KUKA KRL program: wkz2_an.src, wkz2_an.dat

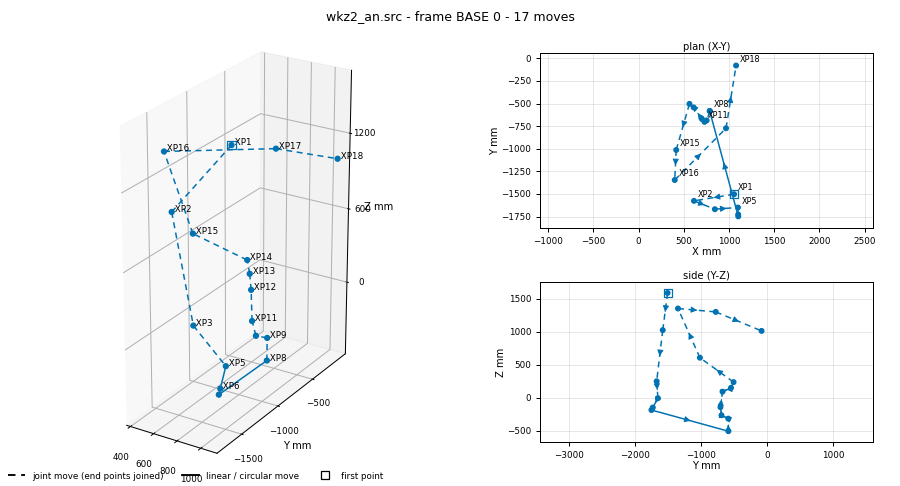
[picture p0: tool path of wkz2_an.src in frame BASE 0, 17 of 17 moves have a stored position in this frame; points joined in program order, loops and branches not executed]
--- wkz2_an.src ---
&ACCESS RVO2
&REL 264
&COMMENT PEGA_GRIPPER_ACTROS
&PARAM DISKPATH = Program/WKZ
DEF WKZ2_AN ( )

;FOLD INI
  ;FOLD BASISTECH INI
    GLOBAL INTERRUPT DECL 3 WHEN $STOPMESS==TRUE DO IR_STOPM ( )
    INTERRUPT ON 3
    BAS (#INITMOV,0 )
  ;ENDFOLD (BASISTECH INI)
  ;FOLD USER INI
    ;Make your modifications here
  ;ENDFOLD (USER INI)
;ENDFOLD (INI)
; Caracterização dos meios de produção:
; Versão Atual:10/06/2015
; Name: P13.090-R6 CHANGES: Pega Garra Actros

CHK_W8_Wechs_OK ( )          ; CHECK FLANGE OK
$ov_pro=50
;FOLD PTP P1 Vel=100 % PDAT1 Tool[8]:Tool Changer Base[0];%{PE}%R 8.2.24,%MKUKATPBASIS,%CMOVE,%VPTP,%P 1:PTP, 2:P1, 3:, 5:100, 7:PDAT1
$BWDSTART=FALSE
PDAT_ACT=PPDAT1
FDAT_ACT=FP1
BAS(#PTP_PARAMS,100)
PTP XP1
;ENDFOLD

;FOLD WAIT FOR ( IN 169 'DEPOSITO 2 OCUPADO' );%{PE}%R 8.2.24,%MKUKATPBASIS,%CEXT_WAIT_FOR,%VEXT_WAIT_FOR,%P 2:, 4:, 5:$IN, 6:169, 7:DEPOSITO 2 OCUPADO, 9:
WAIT FOR  ( $IN[169] )
;ENDFOLD
;FOLD WAIT FOR ( NOT IN 219 'PLACA DE SUPORTE FUNDIDA' );%{PE}%R 8.2.24,%MKUKATPBASIS,%CEXT_WAIT_FOR,%VEXT_WAIT_FOR,%P 2:, 4:NOT, 5:$IN, 6:219, 7:PLACA DE SUPORTE FUNDIDA, 9:
WAIT FOR  (  NOT $IN[219] )
;ENDFOLD
;FOLD PULSE 175 '' State=TRUE Time=0.3 sec;%{PE}%R 8.2.24,%MKUKATPBASIS,%COUT,%VPULSE,%P 2:175, 3:, 5:TRUE, 6:, 8:0.3
PULSE($OUT[175], TRUE,0.3)
;ENDFOLD

;FOLD PTP P2 Vel=100 % PDAT2 Tool[8]:Tool Changer Base[0];%{PE}%R 8.2.24,%MKUKATPBASIS,%CMOVE,%VPTP,%P 1:PTP, 2:P2, 3:, 5:100, 7:PDAT2
$BWDSTART=FALSE
PDAT_ACT=PPDAT2
FDAT_ACT=FP2
BAS(#PTP_PARAMS,100)
PTP XP2
;ENDFOLD

;FOLD WAIT FOR ( IN 173 'PROTECAO DE PINCA ABERTA' );%{PE}%R 8.2.24,%MKUKATPBASIS,%CEXT_WAIT_FOR,%VEXT_WAIT_FOR,%P 2:, 4:, 5:$IN, 6:173, 7:PROTECAO DE PINCA ABERTA, 9:
WAIT FOR  ( $IN[173] )
;ENDFOLD
;FOLD WAIT FOR ( NOT IN 174 'PROTECAO DE PINCA FECHADA' );%{PE}%R 8.2.24,%MKUKATPBASIS,%CEXT_WAIT_FOR,%VEXT_WAIT_FOR,%P 2:, 4:NOT, 5:$IN, 6:174, 7:PROTECAO DE PINCA FECHADA, 9:
WAIT FOR  (  NOT $IN[174] )
;ENDFOLD
;FOLD OUT 223 'DESBLOQUEIA MPS' State=FALSE ;%{PE}%R 8.2.24,%MKUKATPBASIS,%COUT,%VOUTX,%P 2:223, 3:DESBLOQUEIA MPS, 5:FALSE, 6:
$OUT[223]=FALSE
;ENDFOLD
;FOLD OUT 224 'BLOQUEIA MPS' State=TRUE ;%{PE}%R 8.2.24,%MKUKATPBASIS,%COUT,%VOUTX,%P 2:224, 3:BLOQUEIA MPS, 5:TRUE, 6:
$OUT[224]=TRUE
;ENDFOLD

;FOLD PTP P3 Vel=100 % PDAT3 Tool[8]:Tool Changer Base[0];%{PE}%R 8.2.24,%MKUKATPBASIS,%CMOVE,%VPTP,%P 1:PTP, 2:P3, 3:, 5:100, 7:PDAT3
$BWDSTART=FALSE
PDAT_ACT=PPDAT3
FDAT_ACT=FP3
BAS(#PTP_PARAMS,100)
PTP XP3
;ENDFOLD
;FOLD PTP P5 Vel=100 % PDAT5 Tool[8]:Tool Changer Base[0];%{PE}%R 8.2.24,%MKUKATPBASIS,%CMOVE,%VPTP,%P 1:PTP, 2:P5, 3:, 5:100, 7:PDAT5
$BWDSTART=FALSE
PDAT_ACT=PPDAT5
FDAT_ACT=FP5
BAS(#PTP_PARAMS,100)
PTP XP5
;ENDFOLD
;FOLD LIN P6 Vel=0.25 m/s CPDAT1 Tool[8]:Tool Changer Base[0];%{PE}%R 8.2.24,%MKUKATPBASIS,%CMOVE,%VLIN,%P 1:LIN, 2:P6, 3:, 5:0.25, 7:CPDAT1
$BWDSTART=FALSE
LDAT_ACT=LCPDAT1
FDAT_ACT=FP6
BAS(#CP_PARAMS,0.25)
LIN XP6
;ENDFOLD

;FOLD WAIT FOR ( IN 222 'KLASCHKA ATIVADO' );%{PE}%R 8.2.24,%MKUKATPBASIS,%CEXT_WAIT_FOR,%VEXT_WAIT_FOR,%P 2:, 4:, 5:$IN, 6:222, 7:KLASCHKA ATIVADO, 9:
WAIT FOR  ( $IN[222] )
;ENDFOLD
;FOLD OUT 223 'DESBLOQUEIA MPS' State=TRUE ;%{PE}%R 8.2.24,%MKUKATPBASIS,%COUT,%VOUTX,%P 2:223, 3:DESBLOQUEIA MPS, 5:TRUE, 6:
$OUT[223]=TRUE
;ENDFOLD
;FOLD OUT 224 'BLOQUEIA MPS' State=FALSE ;%{PE}%R 8.2.24,%MKUKATPBASIS,%COUT,%VOUTX,%P 2:224, 3:BLOQUEIA MPS, 5:FALSE, 6:
$OUT[224]=FALSE
;ENDFOLD

;FOLD WAIT FOR ( IN 217 'MPS DESTRAVADO' );%{PE}%R 8.2.24,%MKUKATPBASIS,%CEXT_WAIT_FOR,%VEXT_WAIT_FOR,%P 2:, 4:, 5:$IN, 6:217, 7:MPS DESTRAVADO, 9:
WAIT FOR  ( $IN[217] )
;ENDFOLD
;FOLD WAIT FOR ( NOT IN 221 'MPS TRAVADO' );%{PE}%R 8.2.24,%MKUKATPBASIS,%CEXT_WAIT_FOR,%VEXT_WAIT_FOR,%P 2:, 4:NOT, 5:$IN, 6:221, 7:MPS TRAVADO, 9:
WAIT FOR  (  NOT $IN[221] )
;ENDFOLD

;FOLD ; Ponto de pega da ferramenta;%{PE}%R 8.2.24,%MKUKATPBASIS,%CCOMMENT,%VNORMAL,%P 2:Ponto  de  pega  da  ferramenta
;ENDFOLD
;FOLD LIN P7 Vel=0.1 m/s CPDAT2 Tool[8]:Tool Changer Base[0];%{PE}%R 8.2.24,%MKUKATPBASIS,%CMOVE,%VLIN,%P 1:LIN, 2:P7, 3:, 5:0.1, 7:CPDAT2
$BWDSTART=FALSE
LDAT_ACT=LCPDAT2
FDAT_ACT=FP7
BAS(#CP_PARAMS,0.1)
LIN XP7
;ENDFOLD

;FOLD WAIT FOR ( IN 219 'PLACA DE SUPORTE FUNDIDA' );%{PE}%R 8.2.24,%MKUKATPBASIS,%CEXT_WAIT_FOR,%VEXT_WAIT_FOR,%P 2:, 4:, 5:$IN, 6:219, 7:PLACA DE SUPORTE FUNDIDA, 9:
WAIT FOR  ( $IN[219] )
;ENDFOLD
;FOLD OUT 223 'DESBLOQUEIA MPS' State=FALSE ;%{PE}%R 8.2.24,%MKUKATPBASIS,%COUT,%VOUTX,%P 2:223, 3:DESBLOQUEIA MPS, 5:FALSE, 6:
$OUT[223]=FALSE
;ENDFOLD
;FOLD OUT 224 'BLOQUEIA MPS' State=TRUE ;%{PE}%R 8.2.24,%MKUKATPBASIS,%COUT,%VOUTX,%P 2:224, 3:BLOQUEIA MPS, 5:TRUE, 6:
$OUT[224]=TRUE
;ENDFOLD
;FOLD WAIT FOR ( NOT IN 217 'MPS DESTRAVADO' );%{PE}%R 8.2.24,%MKUKATPBASIS,%CEXT_WAIT_FOR,%VEXT_WAIT_FOR,%P 2:, 4:NOT, 5:$IN, 6:217, 7:MPS DESTRAVADO, 9:
WAIT FOR  (  NOT $IN[217] )
;ENDFOLD
;FOLD WAIT FOR ( IN 221 'MPS TRAVADO' );%{PE}%R 8.2.24,%MKUKATPBASIS,%CEXT_WAIT_FOR,%VEXT_WAIT_FOR,%P 2:, 4:, 5:$IN, 6:221, 7:MPS TRAVADO, 9:
WAIT FOR  ( $IN[221] )
;ENDFOLD
;FOLD WAIT Time=1 sec;%{PE}%R 8.2.24,%MKUKATPBASIS,%CWAIT,%VWAIT,%P 3:1
WAIT SEC 1
;ENDFOLD

;FOLD IBUS ON SEGMENT_4;%{PE}%R 8.2.24,%MKUKATPBASIS,%CIBUS,%VMAP,%P 2:#ON, 3:4
$IBUS_ON=IBUS_SEGMENT[4]
$IBUS_OFF=0
;ENDFOLD

;FOLD LIN P8 Vel=0.25 m/s CPDAT3 Tool[2]:Gripper Parabrisa Actro Base[0];%{PE}%R 8.2.24,%MKUKATPBASIS,%CMOVE,%VLIN,%P 1:LIN, 2:P8, 3:, 5:0.25, 7:CPDAT3
$BWDSTART=FALSE
LDAT_ACT=LCPDAT3
FDAT_ACT=FP8
BAS(#CP_PARAMS,0.25)
LIN XP8
;ENDFOLD

;FOLD WAIT FOR ( NOT IN 169 'DEPOSITO 2 OCUPADO' );%{PE}%R 8.2.24,%MKUKATPBASIS,%CEXT_WAIT_FOR,%VEXT_WAIT_FOR,%P 2:, 4:NOT, 5:$IN, 6:169, 7:DEPOSITO 2 OCUPADO, 9:
WAIT FOR  (  NOT $IN[169] )
;ENDFOLD
;FOLD WAIT FOR ( IN 219 'PLACA DE SUPORTE FUNDIDA' );%{PE}%R 8.2.24,%MKUKATPBASIS,%CEXT_WAIT_FOR,%VEXT_WAIT_FOR,%P 2:, 4:, 5:$IN, 6:219, 7:PLACA DE SUPORTE FUNDIDA, 9:
WAIT FOR  ( $IN[219] )
;ENDFOLD

;FOLD ; SETAR GRUPO DE GRAMPOS 1 A 4 CLOSE;%{PE}%R 8.2.24,%MKUKATPBASIS,%CCOMMENT,%VNORMAL,%P 2:SETAR  GRUPO  DE  GRAMPOS  1  A  4 CLOSE
;ENDFOLD
;FOLD SET GRP 1 State=CLO GDAT1;%{PE}%R 8.2.4,%MKUKATPGRP,%CGRP,%VGRP,%P 2:1, 4:1, 5:#NO, 6:GDAT1, 8:0, 10:0
H50(GRP,1,1,GGDAT1)
;ENDFOLD
;FOLD SET GRP 2 State=CLO GDAT2;%{PE}%R 8.2.4,%MKUKATPGRP,%CGRP,%VGRP,%P 2:2, 4:1, 5:#NO, 6:GDAT2, 8:0, 10:0
H50(GRP,2,1,GGDAT2)
;ENDFOLD
;FOLD SET GRP 3 State=CLO GDAT3;%{PE}%R 8.2.4,%MKUKATPGRP,%CGRP,%VGRP,%P 2:3, 4:1, 5:#NO, 6:GDAT3, 8:0, 10:0
H50(GRP,3,1,GGDAT3)
;ENDFOLD
;FOLD SET GRP 4 State=CLO GDAT4;%{PE}%R 8.2.4,%MKUKATPGRP,%CGRP,%VGRP,%P 2:4, 4:1, 5:#NO, 6:GDAT4, 8:0, 10:0
H50(GRP,4,1,GGDAT4)
;ENDFOLD

;FOLD ; CHECAR SE GRAMPOS ESTAO FECHADOS;%{PE}%R 8.2.24,%MKUKATPBASIS,%CCOMMENT,%VNORMAL,%P 2:CHECAR  SE  GRAMPOS  ESTAO  FECHADOS
;ENDFOLD
chk_w2_grp1_clo ()
chk_w2_grp2_clo ()
chk_w2_grp3_clo ()
chk_w2_grp4_clo ()

;FOLD PTP P9 Vel=50 % PDAT6 Tool[2]:Gripper Parabrisa Actro Base[0];%{PE}%R 8.2.24,%MKUKATPBASIS,%CMOVE,%VPTP,%P 1:PTP, 2:P9, 3:, 5:50, 7:PDAT6
$BWDSTART=FALSE
PDAT_ACT=PPDAT6
FDAT_ACT=FP9
BAS(#PTP_PARAMS,50)
PTP XP9
;ENDFOLD
;FOLD PTP P10 Vel=50 % PDAT7 Tool[2]:Gripper Parabrisa Actro Base[0];%{PE}%R 8.2.24,%MKUKATPBASIS,%CMOVE,%VPTP,%P 1:PTP, 2:P10, 3:, 5:50, 7:PDAT7
$BWDSTART=FALSE
PDAT_ACT=PPDAT7
FDAT_ACT=FP10
BAS(#PTP_PARAMS,50)
PTP XP10
;ENDFOLD
;FOLD PTP P11 Vel=50 % PDAT8 Tool[2]:Gripper Parabrisa Actro Base[0];%{PE}%R 8.2.24,%MKUKATPBASIS,%CMOVE,%VPTP,%P 1:PTP, 2:P11, 3:, 5:50, 7:PDAT8
$BWDSTART=FALSE
PDAT_ACT=PPDAT8
FDAT_ACT=FP11
BAS(#PTP_PARAMS,50)
PTP XP11
;ENDFOLD
;FOLD PTP P12 Vel=50 % PDAT9 Tool[2]:Gripper Parabrisa Actro Base[0];%{PE}%R 8.2.24,%MKUKATPBASIS,%CMOVE,%VPTP,%P 1:PTP, 2:P12, 3:, 5:50, 7:PDAT9
$BWDSTART=FALSE
PDAT_ACT=PPDAT9
FDAT_ACT=FP12
BAS(#PTP_PARAMS,50)
PTP XP12
;ENDFOLD
;FOLD PTP P13 Vel=50 % PDAT10 Tool[2]:Gripper Parabrisa Actro Base[0];%{PE}%R 8.2.24,%MKUKATPBASIS,%CMOVE,%VPTP,%P 1:PTP, 2:P13, 3:, 5:50, 7:PDAT10
$BWDSTART=FALSE
PDAT_ACT=PPDAT10
FDAT_ACT=FP13
BAS(#PTP_PARAMS,50)
PTP XP13
;ENDFOLD
;FOLD PTP P14 Vel=50 % PDAT11 Tool[2]:Gripper Parabrisa Actro Base[0];%{PE}%R 8.2.24,%MKUKATPBASIS,%CMOVE,%VPTP,%P 1:PTP, 2:P14, 3:, 5:50, 7:PDAT11
$BWDSTART=FALSE
PDAT_ACT=PPDAT11
FDAT_ACT=FP14
BAS(#PTP_PARAMS,50)
PTP XP14
;ENDFOLD
;FOLD PTP P15 Vel=50 % PDAT12 Tool[2]:Gripper Parabrisa Actro Base[0];%{PE}%R 8.2.24,%MKUKATPBASIS,%CMOVE,%VPTP,%P 1:PTP, 2:P15, 3:, 5:50, 7:PDAT12
$BWDSTART=FALSE
PDAT_ACT=PPDAT12
FDAT_ACT=FP15
BAS(#PTP_PARAMS,50)
PTP XP15
;ENDFOLD
;FOLD PTP P16 CONT Vel=50 % PDAT13 Tool[2]:Gripper Parabrisa Actro Base[0];%{PE}%R 8.2.24,%MKUKATPBASIS,%CMOVE,%VPTP,%P 1:PTP, 2:P16, 3:C_PTP, 5:50, 7:PDAT13
$BWDSTART=FALSE
PDAT_ACT=PPDAT13
FDAT_ACT=FP16
BAS(#PTP_PARAMS,50)
PTP XP16 C_PTP
;ENDFOLD
;FOLD PTP P17 CONT Vel=50 % PDAT14 Tool[2]:Gripper Parabrisa Actro Base[0];%{PE}%R 8.2.24,%MKUKATPBASIS,%CMOVE,%VPTP,%P 1:PTP, 2:P17, 3:C_PTP, 5:50, 7:PDAT14
$BWDSTART=FALSE
PDAT_ACT=PPDAT14
FDAT_ACT=FP17
BAS(#PTP_PARAMS,50)
PTP XP17 C_PTP
;ENDFOLD
;FOLD PTP P18 Vel=50 % PDAT15 Tool[2]:Gripper Parabrisa Actro Base[0];%{PE}%R 8.2.24,%MKUKATPBASIS,%CMOVE,%VPTP,%P 1:PTP, 2:P18, 3:, 5:50, 7:PDAT15
$BWDSTART=FALSE
PDAT_ACT=PPDAT15
FDAT_ACT=FP18
BAS(#PTP_PARAMS,50)
PTP XP18
;ENDFOLD

;FOLD ; SETAR GRUPO DE GRAMPOS 1 A 4 OPEN;%{PE}%R 8.2.24,%MKUKATPBASIS,%CCOMMENT,%VNORMAL,%P 2:SETAR  GRUPO  DE  GRAMPOS  1  A  4 OPEN
;ENDFOLD
;FOLD SET GRP 1 State=OPN GDAT5;%{PE}%R 8.2.4,%MKUKATPGRP,%CGRP,%VGRP,%P 2:1, 4:2, 5:#NO, 6:GDAT5, 8:0, 10:0
H50(GRP,1,2,GGDAT5)
;ENDFOLD
;FOLD SET GRP 2 State=OPN GDAT6;%{PE}%R 8.2.4,%MKUKATPGRP,%CGRP,%VGRP,%P 2:2, 4:2, 5:#NO, 6:GDAT6, 8:0, 10:0
H50(GRP,2,2,GGDAT6)
;ENDFOLD
;FOLD SET GRP 3 State=OPN GDAT7;%{PE}%R 8.2.4,%MKUKATPGRP,%CGRP,%VGRP,%P 2:3, 4:2, 5:#NO, 6:GDAT7, 8:0, 10:0
H50(GRP,3,2,GGDAT7)
;ENDFOLD
;FOLD SET GRP 4 State=OPN GDAT9;%{PE}%R 8.2.4,%MKUKATPGRP,%CGRP,%VGRP,%P 2:4, 4:2, 5:#NO, 6:GDAT9, 8:0, 10:0
H50(GRP,4,2,GGDAT9)
;ENDFOLD
$ov_pro=100
chk_w2_grp1_opn ()
chk_w2_grp2_opn ()
chk_w2_grp3_opn ()
chk_w2_grp4_opn ()

;FOLD WAIT FOR ( IN 3339 'AGUARDA AGV NA POSICAO' );%{PE}%R 8.2.24,%MKUKATPBASIS,%CEXT_WAIT_FOR,%VEXT_WAIT_FOR,%P 2:, 4:, 5:$IN, 6:3339, 7:AGUARDA AGV NA POSICAO, 9:
WAIT FOR  ( $IN[3339] )
;ENDFOLD

END

--- wkz2_an.dat ---
&ACCESS RVO2
&REL 264
&COMMENT PEGA_GRIPPER_ACTROS
&PARAM DISKPATH = Program/WKZ
DEFDAT  wkz2_an
;FOLD EXTERNAL DECLARATIONS;%{PE}%MKUKATPBASIS,%CEXT,%VCOMMON,%P
;FOLD BASISTECH EXT;%{PE}%MKUKATPBASIS,%CEXT,%VEXT,%P
EXT  BAS (BAS_COMMAND  :IN,REAL  :IN )
DECL INT SUCCESS
;ENDFOLD (BASISTECH EXT)
;FOLD USER EXT;%{E}%MKUKATPUSER,%CEXT,%VEXT,%P
;Make your modifications here
;ENDFOLD (USER EXT)
;ENDFOLD (EXTERNAL DECLARATIONS)

;# ============ START PATH : wkz2_an =============
DECL FDAT Fnew_wkz2_an_p44={TOOL_NO 8,BASE_NO 0,IPO_FRAME #BASE,POINT2[] " "}
DECL PDAT PP_OLP1={VEL 100.0,ACC 50.0,APO_DIST 0.0}
DECL E6POS Xnew_wkz2_an_p44={X 612.940979,Y -1576.12097,Z 1025.58899,A -56.8068008,B -30.1534004,C 157.338699,S 2,T 2}
DECL FDAT Fnew_wkz2_an_p16={TOOL_NO 8,BASE_NO 0,IPO_FRAME #BASE,POINT2[] " "}
DECL PDAT PP_OLP2={VEL 100.0,ACC 100.0,APO_DIST 0.0}
DECL E6POS Xnew_wkz2_an_p16={X 843.835999,Y -1668.32202,Z 250.856995,A -56.8068008,B -30.1534004,C 157.338699,S 2,T 2}
DECL FDAT Fnew_wkz2_an_p17={TOOL_NO 8,BASE_NO 0,IPO_FRAME #BASE,POINT2[] " "}
DECL PDAT PP_OLP3={VEL 100.0,ACC 100.0,APO_DIST 0.0}
DECL E6POS Xnew_wkz2_an_p17={X 1098.79395,Y -1649.33801,Z -5.05700016,A -73.2769012,B -27.9207001,C 173.073105,S 2,T 2}
DECL FDAT Fnew_wkz2_an_p4={TOOL_NO 8,BASE_NO 0,IPO_FRAME #BASE,POINT2[] " "}
DECL E6POS Xnew_wkz2_an_p4={X 1101.74304,Y -1726.75305,Z -146.546005,A -73.2770996,B -27.9211998,C 173.073196,S 2,T 2}
DECL LDAT LL_OLP1={VEL 0.25,ACC 100.0,APO_DIST 0.0,APO_FAC 0.0,ORI_TYP #VAR,CIRC_TYP #BASE,JERK_FAC 50.0}
DECL FDAT Fnew_wkz2_an_p5={TOOL_NO 8,BASE_NO 0,IPO_FRAME #BASE,POINT2[] " "}
DECL E6POS Xnew_wkz2_an_p5={X 1102.474,Y -1745.90198,Z -181.546005,A -73.2769012,B -27.9209003,C 173.073105,S 2,T 2}
DECL LDAT LL_OLP2={VEL 0.100000001,ACC 100.0,APO_DIST 0.0,APO_FAC 0.0,ORI_TYP #VAR,CIRC_TYP #BASE,JERK_FAC 50.0}
DECL FDAT Fnew_wkz2_an_p11={TOOL_NO 2,BASE_NO 0,IPO_FRAME #BASE,POINT2[] " "}
DECL E6POS Xnew_wkz2_an_p11={X 786.29303,Y -582.55603,Z -504.964996,A 0.253399998,B -1.02199996,C -179.584305,S 2,T 2}
DECL LDAT LL_OLP3={VEL 0.25,ACC 100.0,APO_DIST 0.0,APO_FAC 0.0,ORI_TYP #VAR,CIRC_TYP #BASE,JERK_FAC 50.0}
DECL FDAT Fnew_wkz2_an_p12={TOOL_NO 2,BASE_NO 0,IPO_FRAME #BASE,POINT2[] " "}
DECL PDAT PP_OLP4={VEL 100.0,ACC 50.0,APO_DIST 0.0}
DECL E6POS Xnew_wkz2_an_p12={X 788.83197,Y -583.976013,Z -314.804993,A 0.253100008,B -1.0223,C -179.584702,S 2,T 2}
DECL FDAT Fnew_wkz2_an_p13={TOOL_NO 2,BASE_NO 0,IPO_FRAME #BASE,POINT2[] " "}
DECL PDAT PP_OLP5={VEL 100.0,ACC 50.0,APO_DIST 0.0}
DECL E6POS Xnew_wkz2_an_p13={X 753.492004,Y -686.713989,Z -263.341003,A 0.255299985,B -1.02450001,C -179.584595,S 2,T 2}
DECL FDAT Fnew_wkz2_an_p18={TOOL_NO 2,BASE_NO 0,IPO_FRAME #BASE,POINT2[] " "}
DECL PDAT PP_OLP6={VEL 100.0,ACC 100.0,APO_DIST 0.0}
DECL E6POS Xnew_wkz2_an_p18={X 728.877991,Y -702.304993,Z -141.432007,A 0.00469999993,B -0.533699989,C -179.897705,S 2,T 2}
DECL FDAT Fnew_wkz2_an_p33={TOOL_NO 2,BASE_NO 0,IPO_FRAME #BASE,POINT2[] " "}
DECL PDAT PP_OLP7={VEL 100.0,ACC 100.0,APO_DIST 0.0}
DECL E6POS Xnew_wkz2_an_p33={X 702.591003,Y -670.484009,Z -1.97099996,A -0.302599996,B -1.01380002,C -179.617706,S 2,T 2}
DECL FDAT Fnew_wkz2_an_p37={TOOL_NO 2,BASE_NO 0,IPO_FRAME #BASE,POINT2[] " "}
DECL PDAT PP_OLP8={VEL 100.0,ACC 100.0,APO_DIST 0.0}
DECL E6POS Xnew_wkz2_an_p37={X 600.364014,Y -522.731018,Z 51.5839996,A -0.309100002,B -1.0122,C -179.757004,S 2,T 2}
DECL FDAT Fnew_wkz2_an_p38={TOOL_NO 2,BASE_NO 0,IPO_FRAME #BASE,POINT2[] " "}
DECL PDAT PP_OLP9={VEL 100.0,ACC 100.0,APO_DIST 0.0}
DECL E6POS Xnew_wkz2_an_p38={X 562.674011,Y -503.727997,Z 237.981003,A -9.11750031,B -5.62230015,C 153.765503,S 2,T 2}
DECL FDAT Fnew_wkz2_an_p42={TOOL_NO 2,BASE_NO 0,IPO_FRAME #BASE,POINT2[] " "}
DECL PDAT PP_OLP10={VEL 100.0,ACC 100.0,APO_DIST 0.0}
DECL E6POS Xnew_wkz2_an_p42={X 978.356018,Y -287.113007,Z 541.031982,A 9.17619991,B -20.1103001,C 143.3797,S 2,T 2}
DECL FDAT Fnew_wkz2_an_p43={TOOL_NO 2,BASE_NO 0,IPO_FRAME #BASE,POINT2[] " "}
DECL PDAT PP_OLP11={VEL 100.0,ACC 100.0,APO_DIST 0.0}
DECL E6POS Xnew_wkz2_an_p43={X 1078.0,Y -78.862999,Z 664.578003,A 0.512600005,B -24.8574009,C 146.008606,S 2,T 2}
DECL BASIS_SUGG_T LAST_BASIS={POINT1[] "P20                     ",POINT2[] "P20                     ",CP_PARAMS[] "CPDAT3                  ",PTP_PARAMS[] "PDAT17                  ",CONT[] "                        ",CP_VEL[] "0.25                    ",PTP_VEL[] "100                     ",SYNC_PARAMS[] "SYNCDAT                 ",SPL_NAME[] "S0                      "}
DECL E6POS XP1={X 1055.88904,Y -1502.42297,Z 1588.46497,A -71.8623123,B -60.8086586,C 178.730499,S 18,T 2,E1 0.0,E2 0.0,E3 0.0,E4 0.0,E5 0.0,E6 0.0}
DECL FDAT FP1={TOOL_NO 8,BASE_NO 0,IPO_FRAME #BASE,POINT2[] " ",TQ_STATE FALSE}
DECL PDAT PPDAT1={VEL 100.0,ACC 100.0,APO_DIST 100.0,GEAR_JERK 50.0}
DECL E6POS XP2={X 612.938782,Y -1576.11304,Z 1025.57605,A -56.8084106,B -30.1530895,C 157.339798,S 18,T 2,E1 0.0,E2 0.0,E3 0.0,E4 0.0,E5 0.0,E6 0.0}
DECL FDAT FP2={TOOL_NO 8,BASE_NO 0,IPO_FRAME #BASE,POINT2[] " ",TQ_STATE FALSE}
DECL PDAT PPDAT2={VEL 100.0,ACC 100.0,APO_DIST 100.0,GEAR_JERK 50.0}
DECL E6POS XP3={X 843.833618,Y -1668.31494,Z 250.858704,A -56.807251,B -30.1531506,C 157.339203,S 18,T 2,E1 0.0,E2 0.0,E3 0.0,E4 0.0,E5 0.0,E6 0.0}
DECL FDAT FP3={TOOL_NO 8,BASE_NO 0,IPO_FRAME #BASE,POINT2[] " ",TQ_STATE FALSE}
DECL PDAT PPDAT3={VEL 100.0,ACC 50.0,APO_DIST 100.0,GEAR_JERK 50.0}
DECL E6POS XP4={X 1070.15295,Y -1848.78406,Z 103.901703,A -73.2903366,B -27.8212204,C 173.081299,S 18,T 2,E1 0.0,E2 0.0,E3 0.0,E4 0.0,E5 0.0,E6 0.0}
DECL FDAT FP4={TOOL_NO 8,BASE_NO 0,IPO_FRAME #BASE,POINT2[] " ",TQ_STATE FALSE}
DECL PDAT PPDAT4={VEL 100.0,ACC 100.0,APO_DIST 100.0,GEAR_JERK 50.0}
DECL GRP_SUGG_T LAST_GRP={NUMBER[] "4                       ",STATE[] "1                       ",PARAMS[] "GDAT4                   "}
DECL E6POS XP5={X 1098.79602,Y -1649.34802,Z -5.03718805,A -73.2673264,B -27.9203205,C 173.069504,S 18,T 2,E1 0.0,E2 0.0,E3 0.0,E4 0.0,E5 0.0,E6 0.0}
DECL FDAT FP5={TOOL_NO 8,BASE_NO 0,IPO_FRAME #BASE,POINT2[] " ",TQ_STATE FALSE}
DECL PDAT PPDAT5={VEL 100.0,ACC 100.0,APO_DIST 100.0,GEAR_JERK 50.0}
DECL E6POS XP6={X 1101.74097,Y -1726.75598,Z -146.535294,A -73.2780228,B -27.9206905,C 173.074005,S 18,T 2,E1 0.0,E2 0.0,E3 0.0,E4 0.0,E5 0.0,E6 0.0}
DECL FDAT FP6={TOOL_NO 8,BASE_NO 0,IPO_FRAME #BASE,POINT2[] " ",TQ_STATE FALSE}
DECL LDAT LCPDAT1={VEL 2.0,ACC 100.0,APO_DIST 100.0,APO_FAC 50.0,AXIS_VEL 100.0,AXIS_ACC 100.0,ORI_TYP #VAR,CIRC_TYP #BASE,JERK_FAC 50.0,GEAR_JERK 50.0,EXAX_IGN 0}
DECL E6POS XP7={X 1102.50403,Y -1747.31702,Z -184.174393,A -73.2694321,B -27.9181194,C 173.068497,S 18,T 2,E1 0.0,E2 0.0,E3 0.0,E4 0.0,E5 0.0,E6 0.0}
DECL FDAT FP7={TOOL_NO 8,BASE_NO 0,IPO_FRAME #BASE,POINT2[] " ",TQ_STATE FALSE}
DECL LDAT LCPDAT2={VEL 2.0,ACC 100.0,APO_DIST 100.0,APO_FAC 50.0,AXIS_VEL 100.0,AXIS_ACC 100.0,ORI_TYP #VAR,CIRC_TYP #BASE,JERK_FAC 50.0,GEAR_JERK 50.0,EXAX_IGN 0}
DECL E6POS XP8={X 786.28833,Y -582.550781,Z -504.954407,A 0.253419489,B -1.02197099,C -179.584,S 18,T 2,E1 0.0,E2 0.0,E3 0.0,E4 0.0,E5 0.0,E6 0.0}
DECL FDAT FP8={TOOL_NO 2,BASE_NO 0,IPO_FRAME #BASE,POINT2[] " ",TQ_STATE FALSE}
DECL LDAT LCPDAT3={VEL 2.0,ACC 100.0,APO_DIST 100.0,APO_FAC 50.0,AXIS_VEL 100.0,AXIS_ACC 100.0,ORI_TYP #VAR,CIRC_TYP #BASE,JERK_FAC 50.0,GEAR_JERK 50.0,EXAX_IGN 0}
DECL E6POS XP9={X 788.821777,Y -583.967224,Z -314.793488,A 0.253417194,B -1.02216303,C -179.584198,S 18,T 2,E1 0.0,E2 0.0,E3 0.0,E4 0.0,E5 0.0,E6 0.0}
DECL FDAT FP9={TOOL_NO 2,BASE_NO 0,IPO_FRAME #BASE,POINT2[] " ",TQ_STATE FALSE}
DECL PDAT PPDAT6={VEL 100.0,ACC 100.0,APO_DIST 100.0,GEAR_JERK 50.0}
DECL GRP_TYP GCONT={G_APO #YES,GRP_TIME 0.0,CTRL #OFF,DLY 0,DST 0}
DECL E6POS XP10={X 753.30658,Y -686.742981,Z -263.305695,A 0.262432188,B -1.01997399,C -179.584,S 18,T 2,E1 0.0,E2 0.0,E3 0.0,E4 0.0,E5 0.0,E6 0.0}
DECL FDAT FP10={TOOL_NO 2,BASE_NO 0,IPO_FRAME #BASE,POINT2[] " ",TQ_STATE FALSE}
DECL PDAT PPDAT7={VEL 100.0,ACC 50.0,APO_DIST 100.0,GEAR_JERK 50.0}
DECL E6POS XP11={X 728.857788,Y -702.299377,Z -141.422302,A 0.00528541021,B -0.533387423,C -179.897202,S 18,T 2,E1 0.0,E2 0.0,E3 0.0,E4 0.0,E5 0.0,E6 0.0}
DECL FDAT FP11={TOOL_NO 2,BASE_NO 0,IPO_FRAME #BASE,POINT2[] " ",TQ_STATE FALSE}
DECL PDAT PPDAT8={VEL 100.0,ACC 50.0,APO_DIST 100.0,GEAR_JERK 50.0}
DECL E6POS XP12={X 700.793579,Y -670.951172,Z 93.8796005,A -0.304085791,B -1.01611602,C -179.614304,S 18,T 2,E1 0.0,E2 0.0,E3 0.0,E4 0.0,E5 0.0,E6 0.0}
DECL FDAT FP12={TOOL_NO 2,BASE_NO 0,IPO_FRAME #BASE,POINT2[] " ",TQ_STATE FALSE}
DECL PDAT PPDAT9={VEL 100.0,ACC 100.0,APO_DIST 100.0,GEAR_JERK 50.0}
DECL E6POS XP13={X 609.002197,Y -542.534485,Z 151.936707,A -0.474724114,B -0.604779422,C -179.868103,S 18,T 2,E1 0.0,E2 0.0,E3 0.0,E4 0.0,E5 0.0,E6 0.0}
DECL FDAT FP13={TOOL_NO 2,BASE_NO 0,IPO_FRAME #BASE,POINT2[] " ",TQ_STATE FALSE}
DECL PDAT PPDAT10={VEL 100.0,ACC 100.0,APO_DIST 100.0,GEAR_JERK 50.0}
DECL E6POS XP14={X 562.718872,Y -503.715088,Z 237.983398,A -9.11649132,B -5.62477922,C 153.766907,S 18,T 2,E1 0.0,E2 0.0,E3 0.0,E4 0.0,E5 0.0,E6 0.0}
DECL FDAT FP14={TOOL_NO 2,BASE_NO 0,IPO_FRAME #BASE,POINT2[] " ",TQ_STATE FALSE}
DECL PDAT PPDAT11={VEL 100.0,ACC 100.0,APO_DIST 100.0,GEAR_JERK 50.0}
DECL E6POS XP15={X 416.388885,Y -1013.36902,Z 607.772583,A -4.08418417,B -4.78348684,C 150.544098,S 18,T 2,E1 0.0,E2 0.0,E3 0.0,E4 0.0,E5 0.0,E6 0.0}
DECL FDAT FP15={TOOL_NO 2,BASE_NO 0,IPO_FRAME #BASE,POINT2[] " ",TQ_STATE FALSE}
DECL PDAT PPDAT12={VEL 100.0,ACC 100.0,APO_DIST 100.0,GEAR_JERK 50.0}
DECL E6POS XP16={X 400.190887,Y -1345.43701,Z 1352.74597,A 4.42342091,B -14.8097095,C 106.8871,S 18,T 2,E1 0.0,E2 0.0,E3 0.0,E4 0.0,E5 0.0,E6 0.0}
DECL FDAT FP16={TOOL_NO 2,BASE_NO 0,IPO_FRAME #BASE,POINT2[] " ",TQ_STATE FALSE}
DECL PDAT PPDAT13={VEL 100.0,ACC 100.0,APO_DIST 100.0,APO_MODE #CPTP,GEAR_JERK 50.0}
DECL E6POS XP17={X 967.026184,Y -773.494324,Z 1301.31006,A 10.1119204,B -33.0862885,C 128.648895,S 18,T 2,E1 0.0,E2 0.0,E3 0.0,E4 0.0,E5 0.0,E6 0.0}
DECL FDAT FP17={TOOL_NO 2,BASE_NO 0,IPO_FRAME #BASE,POINT2[] " ",TQ_STATE FALSE}
DECL PDAT PPDAT14={VEL 100.0,ACC 100.0,APO_DIST 100.0,APO_MODE #CPTP,GEAR_JERK 50.0}
DECL E6POS XP18={X 1078.36804,Y -79.8228989,Z 1013.84601,A 0.511365473,B -24.8507099,C 145.9991,S 18,T 2,E1 0.0,E2 0.0,E3 0.0,E4 0.0,E5 0.0,E6 0.0}
DECL FDAT FP18={TOOL_NO 2,BASE_NO 0,IPO_FRAME #BASE,POINT2[] " ",TQ_STATE FALSE}
DECL PDAT PPDAT15={VEL 100.0,ACC 100.0,APO_DIST 100.0,GEAR_JERK 50.0}
DECL E6POS XP19={X 786.362122,Y -582.509216,Z -496.813385,A 0.249103606,B -1.02410901,C -179.582306,S 18,T 2,E1 0.0,E2 0.0,E3 0.0,E4 0.0,E5 0.0,E6 0.0}
DECL FDAT FP19={TOOL_NO 2,BASE_NO 0,IPO_FRAME #BASE,POINT2[] " ",TQ_STATE FALSE}
DECL PDAT PPDAT16={VEL 100.0,ACC 100.0,APO_DIST 100.0,GEAR_JERK 50.0}
DECL GRP_TYP GGDAT1={G_APO #NO,GRP_TIME 0.200000003,CTRL #OFF,DLY 0,DST 1}
DECL GRP_TYP GGDAT2={G_APO #NO,GRP_TIME 0.200000003,CTRL #OFF,DLY 0,DST 1}
DECL GRP_TYP GGDAT3={G_APO #NO,GRP_TIME 0.200000003,CTRL #OFF,DLY 0,DST 1}
DECL GRP_TYP GGDAT4={G_APO #NO,GRP_TIME 0.200000003,CTRL #OFF,DLY 0,DST 1}
DECL GRP_TYP GGDAT5={G_APO #NO,GRP_TIME 0.200000003,CTRL #OFF,DLY 0,DST 1}
DECL GRP_TYP GGDAT6={G_APO #NO,GRP_TIME 0.200000003,CTRL #OFF,DLY 0,DST 1}
DECL GRP_TYP GGDAT7={G_APO #NO,GRP_TIME 0.200000003,CTRL #OFF,DLY 0,DST 1}
DECL GRP_TYP GGDAT9={G_APO #NO,GRP_TIME 0.200000003,CTRL #OFF,DLY 0,DST 1}
DECL E6POS XP20={X 1248.69702,Y -1730.67505,Z -1000.89203,A 79.231987,B 73.5589066,C -8.79684162,S 18,T 2,E1 0.0,E2 0.0,E3 0.0,E4 0.0,E5 0.0,E6 0.0}
DECL FDAT FP20={TOOL_NO 4,BASE_NO 0,IPO_FRAME #BASE,POINT2[] " ",TQ_STATE FALSE}
DECL PDAT PPDAT17={VEL 100.0,ACC 100.0,APO_DIST 100.0,GEAR_JERK 50.0}
ENDDAT
